Staubli VAL3: F6_Axis8.pgx

program F6_Axis8()
begin
  call Axis8:onF2Event()
end
